# EPICS autosave request: SMC100XXApp/Db/SMC100XX_settings.req
# Newport SMC100CC/PP settings
$(P)config
$(P)accel
$(P)velocity
$(P)mres
$(P)ustep
$(P)absPos
$(P)relPos
$(P)absPos.DRVH
